(* IEC 61131-3 sources: Openplc_v3/webserver/st_files, 9 files *)

(* ---- 148081.st ---- *)
PROGRAM plc1
  VAR
    ColorSensor_RED AT %IW0 : INT;
    ColorSensor_GREEN AT %IW1 : INT;
    ColorSensor_BLUE AT %IW2 : INT;
    RangeSensor AT %IW3 : INT;
    Pump AT %QX0.4 : BOOL := False;
    treatmentComplete AT %IX100.0 : BOOL := False;
  END_VAR
  VAR
    desiredDistanceFill : REAL := 7.0;
    measuredDistance : REAL;
  END_VAR

  (*Workaround to distance measure bug*)
  measuredDistance := INT_TO_REAL(RangeSensor)/100.0;
  desiredDistanceFill := 7.0;

  IF INT_TO_REAL(RangeSensor) > 99.0 THEN
    treatmentComplete := True;
    PRINT('Treatment is Complete\n');
  ELSE
    treatmentComplete := False;
  END_IF;

  IF treatmentComplete THEN
    IF measuredDistance > desiredDistanceFill THEN
      Pump := TRUE;
    ELSE
      Pump := FALSE;
    END_IF;
  END_IF;

  PRINT('Measured Distance: ', measuredDistance, '\n');
  PRINT('Desired Distance: ', desiredDistanceFill, '\n');
END_PROGRAM

CONFIGURATION Config0

  RESOURCE Res0 ON PLC
    TASK task0(INTERVAL := T#20ms,PRIORITY := 0);
    PROGRAM instance0 WITH task0 : plc1;
  END_RESOURCE
END_CONFIGURATION

(* ---- 333950.st ---- *)
PROGRAM plc1
  VAR
    ColorSensor_RED AT %IW0 : INT;
    ColorSensor_GREEN AT %IW1 : INT;
    ColorSensor_BLUE AT %IW2 : INT;
    RangeSensor AT %IW3 : INT;
    Pump AT %QX0.4 : BOOL := False;
    treatmentComplete AT %IX100.0 : BOOL := False;
  END_VAR
  VAR
    desiredDistanceFill : REAL := 7.0;
    measuredDistance : REAL;
  END_VAR

  (*Workaround to distance measure bug*)
  measuredDistance := INT_TO_REAL(RangeSensor)/100.0;
  desiredDistanceFill := 7.0;

  IF INT_TO_REAL(RangeSensor) > 99.0 THEN
    treatmentComplete := True;
    PRINT('Treatment is Complete\n');
  ELSE
    treatmentComplete := False;
  END_IF;

  IF treatmentComplete THEN
    IF measuredDistance > desiredDistanceFill THEN
      Pump := TRUE;
    ELSE
      Pump := FALSE;
    END_IF;
  END_IF;

  PRINT('Measured Distance: ', measuredDistance, '\n');
  PRINT('Desired Distance: ', desiredDistanceFill, '\n');
END_PROGRAM

CONFIGURATION Config0

  RESOURCE Res0 ON PLC
    TASK task0(INTERVAL := T#20ms,PRIORITY := 0);
    PROGRAM instance0 WITH task0 : plc1;
  END_RESOURCE
END_CONFIGURATION

(* ---- 441230.st ---- *)
PROGRAM plc1
  VAR
    ColorSensor_RED AT %IW0 : INT;
    ColorSensor_GREEN AT %IW1 : INT;
    ColorSensor_BLUE AT %IW2 : INT;
    RangeSensor AT %IW3 : INT;
    Pump AT %QX0.4 : BOOL := False;
    treatmentComplete AT %IX100.0 : BOOL := False;
  END_VAR
  VAR
    desiredDistanceFill : REAL := 7.0;
    measuredDistance : REAL;
  END_VAR

  (*Workaround to distance measure bug*)
  measuredDistance := INT_TO_REAL(RangeSensor)/100.0;
  desiredDistanceFill := 7.0;

  IF INT_TO_REAL(RangeSensor) > 99.0 THEN
    treatmentComplete := True;
  ELSE
    treatmentComplete := False;
  END_IF;

  IF treatmentComplete THEN
          IF measuredDistance > desiredDistanceFill THEN
            Pump := TRUE;
          ELSE
            Pump := FALSE;
          END_IF;
  END_IF;
END_PROGRAM

CONFIGURATION Config0

  RESOURCE Res0 ON PLC
    TASK task0(INTERVAL := T#20ms,PRIORITY := 0);
    PROGRAM instance0 WITH task0 : plc1;
  END_RESOURCE
END_CONFIGURATION

(* ---- 496597.st ---- *)
PROGRAM plc1
  VAR
    ColorSensor_RED AT %IW0 : INT;
    ColorSensor_GREEN AT %IW1 : INT;
    ColorSensor_BLUE AT %IW2 : INT;
    RangeSensor AT %IW3 : INT;
    Pump AT %QX0.4 : BOOL := False;
    treatmentComplete AT %IX100.0 : BOOL := False;
  END_VAR
  VAR
    desiredDistanceFill : REAL := 7.0;
    measuredDistance : REAL;
  END_VAR

  (*Workaround to distance measure bug*)
  measuredDistance := INT_TO_REAL(RangeSensor)/100.0;
  desiredDistanceFill := 7.0;

  IF INT_TO_REAL(RangeSensor) > 99.0 THEN
    treatmentComplete := True;
  ELSE
    treatmentComplete := False;
  END_IF;

  IF treatmentComplete THEN
          IF measuredDistance > desiredDistanceFill THEN
            Pump := TRUE;
          ELSE
            Pump := FALSE;
          END_IF;
  END_IF;
END_PROGRAM

CONFIGURATION Config0

  RESOURCE Res0 ON PLC
    TASK task0(INTERVAL := T#20ms,PRIORITY := 0);
    PROGRAM instance0 WITH task0 : plc1;
  END_RESOURCE
END_CONFIGURATION

(* ---- 705793.st ---- *)
PROGRAM plc1
  VAR
    ColorSensor_RED AT %IW0 : INT;
    ColorSensor_GREEN AT %IW1 : INT;
    ColorSensor_BLUE AT %IW2 : INT;
    RangeSensor AT %IW3 : INT;
    Pump AT %QX0.4 : BOOL := False;
    treatmentComplete AT %IX100.0 : BOOL := False;
  END_VAR
  VAR
    desiredDistanceFill : REAL := 7.0;
    measuredDistance : REAL;
  END_VAR

  (*Workaround to distance measure bug*)
  measuredDistance := INT_TO_REAL(RangeSensor)/100.0;
  desiredDistanceFill := 7.0;

  IF INT_TO_REAL(RangeSensor) > 99.0 THEN
    treatmentComplete := True;
  ELSE
    treatmentComplete := False;
  END_IF;

  IF treatmentComplete THEN
          IF measuredDistance > desiredDistanceFill THEN
            Pump := TRUE;
          ELSE
            Pump := FALSE;
          END_IF;
  END_IF;
END_PROGRAM

CONFIGURATION Config0

  RESOURCE Res0 ON PLC
    TASK task0(INTERVAL := T#20ms,PRIORITY := 0);
    PROGRAM instance0 WITH task0 : plc1;
  END_RESOURCE
END_CONFIGURATION

(* ---- 837052.st ---- *)
PROGRAM plc1
  VAR
    ColorSensor_RED AT %IW0 : INT;
    ColorSensor_GREEN AT %IW1 : INT;
    ColorSensor_BLUE AT %IW2 : INT;
    RangeSensor AT %IW3 : INT;
    Pump AT %QX0.4 : BOOL := False;
    treatmentComplete AT %IX100.0 : BOOL := False;
  END_VAR
  VAR
    desiredDistanceFill : REAL := 7.0;
    measuredDistance : REAL;
  END_VAR

  (*Workaround to distance measure bug*)
  measuredDistance := INT_TO_REAL(RangeSensor)/100.0;
  desiredDistanceFill := 7.0;

  IF treatmentComplete THEN
          IF measuredDistance > desiredDistanceFill THEN
            Pump := TRUE;
          ELSE
            Pump := FALSE;
          END_IF;
  END_IF;
END_PROGRAM

CONFIGURATION Config0

  RESOURCE Res0 ON PLC
    TASK task0(INTERVAL := T#20ms,PRIORITY := 0);
    PROGRAM instance0 WITH task0 : plc1;
  END_RESOURCE
END_CONFIGURATION

(* ---- 901484.st ---- *)
PROGRAM plc1
  VAR
    ColorSensor_RED AT %IW0 : INT;
    ColorSensor_GREEN AT %IW1 : INT;
    ColorSensor_BLUE AT %IW2 : INT;
    RangeSensor AT %IW3 : INT;
    Pump AT %QX0.4 : BOOL := False;
    treatmentComplete AT %IX100.0 : BOOL := False;
  END_VAR
  VAR
    desiredDistanceFill : REAL := 7.0;
    measuredDistance : REAL;
  END_VAR

	PRINT("HELLO")

  (*Workaround to distance measure bug*)
  measuredDistance := INT_TO_REAL(RangeSensor)/100.0;
  desiredDistanceFill := 7.0;

  IF INT_TO_REAL(RangeSensor) > 99.0 THEN
    treatmentComplete := True;
  ELSE
    treatmentComplete := False;
  END_IF;

  IF treatmentComplete THEN
          IF measuredDistance > desiredDistanceFill THEN
            Pump := TRUE;
          ELSE
            Pump := FALSE;
          END_IF;
  END_IF;
END_PROGRAM

CONFIGURATION Config0

  RESOURCE Res0 ON PLC
    TASK task0(INTERVAL := T#20ms,PRIORITY := 0);
    PROGRAM instance0 WITH task0 : plc1;
  END_RESOURCE
END_CONFIGURATION

(* ---- 991605.st ---- *)
PROGRAM plc1
  VAR
    ColorSensor_RED AT %IW0 : INT;
    ColorSensor_GREEN AT %IW1 : INT;
    ColorSensor_BLUE AT %IW2 : INT;
    RangeSensor AT %IW3 : INT;
    Pump AT %QX0.4 : BOOL := False;
    treatmentComplete AT %IX100.0 : BOOL := False;
  END_VAR
  VAR
    desiredDistanceFill : REAL := 7.0;
    measuredDistance : REAL;
  END_VAR

  (*Workaround to distance measure bug*)
  measuredDistance := INT_TO_REAL(RangeSensor)/100.0;
  desiredDistanceFill := 7.0;

  IF INT_TO_REAL(RangeSensor) > 99.0 THEN
    treatmentComplete := True;
  ELSE
    treatmentComplete := False;
  END_IF;

  IF treatmentComplete THEN
          IF measuredDistance > desiredDistanceFill THEN
            Pump := TRUE;
          ELSE
            Pump := FALSE;
          END_IF;
  END_IF;
END_PROGRAM

CONFIGURATION Config0

  RESOURCE Res0 ON PLC
    TASK task0(INTERVAL := T#20ms,PRIORITY := 0);
    PROGRAM instance0 WITH task0 : plc1;
  END_RESOURCE
END_CONFIGURATION

(* ---- blank_program.st ---- *)
PROGRAM prog0
  VAR
    var_in : BOOL;
    var_out : BOOL;
  END_VAR

  var_out := var_in;
END_PROGRAM

CONFIGURATION Config0

  RESOURCE Res0 ON PLC
    TASK Main(INTERVAL := T#50ms,PRIORITY := 0);
    PROGRAM Inst0 WITH Main : prog0;
  END_RESOURCE
END_CONFIGURATION
